{attribute 'qualified_only'}
{attribute 'strict'}
TYPE E_Xbox_Controller_Battery_Types :
(
	// Battery is disconnected
	Disconnected := 0,
	// Battery is wired
	Wired := 1,
	// Battery is alkaline
	Alkaline := 2,
	// Battery is nickel-metal hydride
	NIMH := 3,
	// Battery is unknown
	Unknown := 4
);
END_TYPE

(* stored: Version 1.1.0.1, ProductVersion 3.1.4024.11
   DUT E_Xbox_Controller_Battery_Types: Id {1eac3af5-eade-4890-9e49-5376e579fab8} *)
